TYPE ST_NciAxisIds :
STRUCT
    nX  : UDINT;
    nY  : UDINT;
    nZ  : UDINT;
    nQ1 : UDINT;
    nQ2 : UDINT;
    nQ3 : UDINT;
    nQ4 : UDINT;
    nQ5 : UDINT;
END_STRUCT
END_TYPE

(* stored: Version 1.1.0.1, ProductVersion 3.1.4024.15
   DUT ST_NciAxisIds: Id {0a86367d-0c94-4d22-88c9-189982a2483a} *)
